// TIA Portal V20 export
DATA_BLOCK "ControlNodes"   // DB41
// stored: Access Published, MemoryReserve 100, Namespace Unit1
   VAR
      fuses { ExternalWritable := 'False'} : Struct
         E202Cb480vVoltage24VOK : Bool;   // MotorPowerTripped
         E208Cb480vVoltage24VOK : Bool;   // ReelcutConveyorRingBlowPowerTripped
         E214Cb480vVoltage24VOK : Bool;   // Stacking1ConveyorRingBlowPowerTripped
         E220Cb480vVoltage24VOK : Bool;   // Stacking2ConveyorRingBlowPowerTripped
         E320Cb480vVoltage24VOK : Bool;   // E6404PwsControllerPowerSmpsAcPowerTripped
         E326Cb480vVoltage24VOK : Bool;   // E6704PwsControllerPowerSmpsAcPowerTripped
         E332Cb480vVoltage24VOK : Bool;   // E6804PwsSafetyPowerSmpsAcPowerTripped
         E720Cb480vVoltage24VOK : Bool;   // PowerMeterPowerTripped
         E726CbVoltage24VOK : Bool;   // PowerMeterControlPowerTripped
         E4116Cb480vVoltage24VOK : Bool;   // ProcessorPowerOnTripped
         E4156Cb480vVoltage24VOK : Bool;   // ProgrammingPowerOutletTripped
         E4304CbVoltage24VOK : Bool;   // PanelLedPowerTripped
         E4420CbVoltage24VOK : Bool;   // ControlLevelHubPowerTripped
         E4426CbVoltage24VOK : Bool;   // MainHmiPowerTripped
         E4432CbVoltage24VOK : Bool;   // PortableHmiPowerTripped
         E4456CbVoltage24VOK : Bool;   // PortableHmiPowerTripped
         E5100Cb480vVoltage24VOK : Bool;   // 120VacControlPowerTrPrimaryTripped
         E5110CbVoltage24VOK : Bool;   // 120VacControlPowerTrSecondaryTripped
         E5116CbVoltage24VOK : Bool;   // ControlPowerOnTripped
         E5160CbVoltage24VOK : Bool;   // VisionMonitorPowerStripOutletPowerTripped
         E5166CbVoltage24VOK : Bool;   // McuRfidHandyPowerStripOutletPowerTripped
         E5172CbVoltage24VOK : Bool;   // VisionLightControllerPowerStripOutletPowerTripped
         E5222CbVoltage24VOK : Bool;   // FfuPower1PowerTripped
         E6154CbVoltage24VOK : Bool;   // Et200MpIoOutputPowerTripped
         E6180CbVoltage24VOK : Bool;   // JunctionBoxControlPowerTripped
         E6204CbVoltage24VOK : Bool;   // Class2SmpsPowerTripped
         E6206CbVoltage24VOK : Bool;   // Class2SmpsMonitoringTripped
         E6220CbVoltage24VOK : Bool;   // Et200EcoPn1PowerTripped
         E6224CbVoltage24VOK : Bool;   // Et200EcoPn2PowerTripped
         E6228CbVoltage24VOK : Bool;   // Et200EcoPn3PowerTripped
         E6304CbVoltage24VOK : Bool;   // PanelFanPowerTripped
         E6406CbVoltage24VOK : Bool;   // ControllerDcPowerTripped
         E6416CbVoltage24VOK : Bool;   // ServoControlPowerTripped
         E6422CbVoltage24VOK : Bool;   // Manifold1ControlPowerTripped
         E6456CbVoltage24VOK : Bool;   // RfidPowerTripped
         E6462CbVoltage24VOK : Bool;   // QrReaderPowerTripped
         E6468CbVoltage24VOK : Bool;   // QrReaderPowerTripped
         E6706CbVoltage24VOK : Bool;   // ControllerDcPowerTripped
         E6716CbVoltage24VOK : Bool;   // HandyQrReaderPowerTripped
         E6722CbVoltage24VOK : Bool;   // VisionControllerPowerTripped
         E6728CbVoltage24VOK : Bool;   // LineLaserModule1PowerTripped
         E6734CbVoltage24VOK : Bool;   // LineLaserModule2PowerTripped
         E6756CbVoltage24VOK : Bool;   // EpcController1PowerTripped
         E6762CbVoltage24VOK : Bool;   // EpcController2PowerTripped
         E6768CbVoltage24VOK : Bool;   // EpcController3PowerTripped
         E6774CbVoltage24VOK : Bool;   // DriveCliqHubPowerTripped
         E6780CbVoltage24VOK : Bool;   // EquipmentLedPowerTripped
         E6786CbVoltage24VOK : Bool;   // MotorPowerMcCoilPowerTripped
         E6806CbVoltage24VOK : Bool;   // SafetyDcPowerTripped
         E6816CbVoltage24VOK : Bool;   // Et200SpIoSafetyPowerTripped
         E6836CbVoltage24VOK : Bool;   // JunctionBoxControlPowerTripped
         E6856CbVoltage24VOK : Bool;   // Et200EcoPnSafetyT1PowerTripped
         E110CbVoltage24VOK : Bool;   // MainHMIPowerTrpped
         E156CbVoltage24VOK : Bool;   // ControlDcPowerTripped
         E218CbVoltage24VOK : Bool;   // SafetyDcPowerTripped
      END_STRUCT;
      pws { ExternalWritable := 'False'} : Struct
         powerSupplyE4404PwsOK : Bool;   // PlcPowerSmpsDcOk
         powerSupplyE6104PwsOK : Bool;   // ControlPowerSmpsDcOk
         powerSupplyE6404PwsOK : Bool;   // ControllerPowerSmpsDcOk
         powerSupplyE6704PwsOK : Bool;   // ControllerPowerSmpsDcOk
         powerSupplyE6804PwsOK : Bool;   // SafetyPowerSmpsDcOk
      END_STRUCT;
      motorPowerMC { ExternalWritable := 'False'} : Struct
         FeedBack : Bool;
         McOn : Bool;
         Ready : Bool;
         Operation : Bool;
         Run : Bool;
         Fault : Bool;
         Error : Bool;
      END_STRUCT;
      airOK { ExternalWritable := 'False'} : Bool;   // Compressed air OK
      InitializeEnable { ExternalWritable := 'False'} : Bool;
      AutoStartEnable { ExternalWritable := 'False'} : Bool;
      cmFFU { ExternalWritable := 'False'} : "LER_typeLIU117ControlNode";
      citiMap : "LER_OEM_Data";
      "========Communication========" : Bool;
      BA030 { ExternalWritable := 'False'} : "LER_typeCommunicationControlNode";
      BA040 { ExternalWritable := 'False'} : "LER_typeCommunicationControlNode";
   END_VAR
BEGIN
END_DATA_BLOCK
